FUNCTION_BLOCK Q_Attribute (* Command change attribute( Part 6 - F.38 ) *)
  (* Standard: ISO 11783-6; Description: This command is used to change any attribute with an assigned AID. This message cannot be used to change strings. Return values iso_s16 - E_NO_ERR - OK - E_OVERFLOW - buffer overflow - E_NOACT - Command not possible in current state - E_NO_INSTANCE - No VT client available *)
  (* Version 1.0, 2022-07-08, franz *)
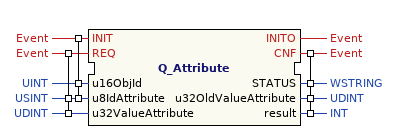
  EVENT_INPUT
    INIT WITH u16ObjId, u8IdAttribute; (* Service Initialization *)
    REQ WITH u8IdAttribute, u32ValueAttribute; (* Service Request *)
  END_EVENT
  EVENT_OUTPUT
    INITO; (* Initialization Confirm *)
    CNF WITH STATUS, u32OldValueAttribute, result, u32OldValueAttribute; (* Confirmation of Requested Service *)
  END_EVENT
  VAR_INPUT
    u16ObjId : UINT; (* Object ID *)
    u8IdAttribute : USINT; (* Attribute ID (AID) - see description of wished object *)
    u32ValueAttribute : UDINT; (* New value for attribute *)
  END_VAR
  VAR_OUTPUT
    STATUS : WSTRING; (* Service Status *)
    u32OldValueAttribute : UDINT; (* Old value for attribute *)
    result : INT; (* retval see description *)
  END_VAR
END_FUNCTION_BLOCK
